// Mitsubishi GX Developer project: 12-201_1204051130   PLC: FX1N

PROGRAM MAIN
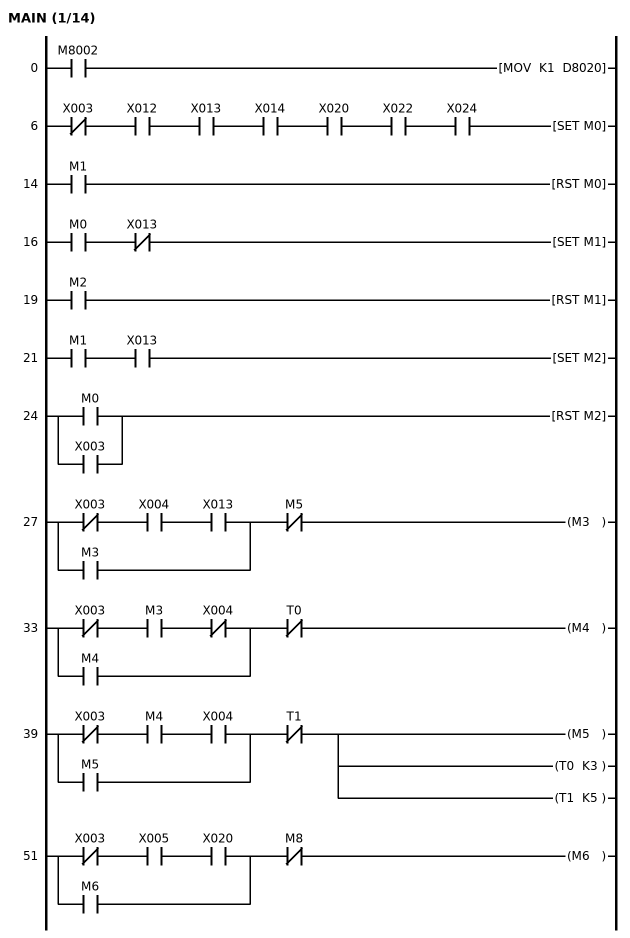
0     LD      M8002
      MOV     K1 D8020
6     LDI     X003
      AND     X012
      AND     X013
      AND     X014
      AND     X020
      AND     X022
      AND     X024
      SET     M0
14    LD      M1
      RST     M0
16    LD      M0
      ANI     X013
      SET     M1
19    LD      M2
      RST     M1
21    LD      M1
      AND     X013
      SET     M2
24    LD      M0
      OR      X003
      RST     M2
27    LDI     X003
      AND     X004
      AND     X013
      OR      M3
      ANI     M5
      OUT     M3
33    LDI     X003
      AND     M3
      ANI     X004
      OR      M4
      ANI     T0
      OUT     M4
39    LDI     X003
      AND     M4
      AND     X004
      OR      M5
      ANI     T1
      OUT     M5
      OUT     T0 K3
      OUT     T1 K5
51    LDI     X003
      AND     X005
      AND     X020
      OR      M6
      ANI     M8
      OUT     M6
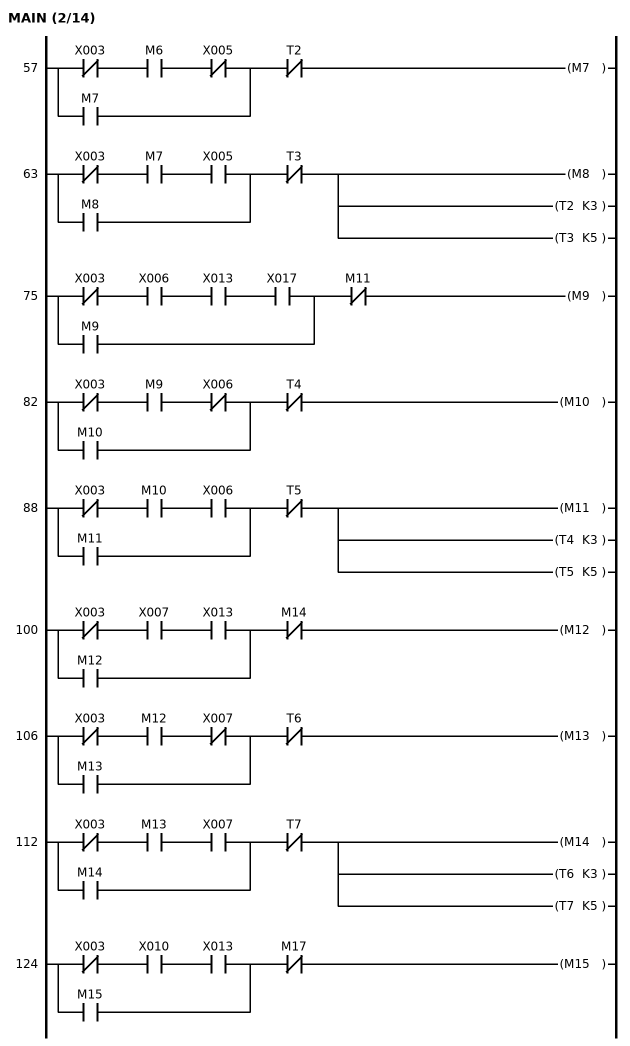
57    LDI     X003
      AND     M6
      ANI     X005
      OR      M7
      ANI     T2
      OUT     M7
63    LDI     X003
      AND     M7
      AND     X005
      OR      M8
      ANI     T3
      OUT     M8
      OUT     T2 K3
      OUT     T3 K5
75    LDI     X003
      AND     X006
      AND     X013
      AND     X017
      OR      M9
      ANI     M11
      OUT     M9
82    LDI     X003
      AND     M9
      ANI     X006
      OR      M10
      ANI     T4
      OUT     M10
88    LDI     X003
      AND     M10
      AND     X006
      OR      M11
      ANI     T5
      OUT     M11
      OUT     T4 K3
      OUT     T5 K5
100   LDI     X003
      AND     X007
      AND     X013
      OR      M12
      ANI     M14
      OUT     M12
106   LDI     X003
      AND     M12
      ANI     X007
      OR      M13
      ANI     T6
      OUT     M13
112   LDI     X003
      AND     M13
      AND     X007
      OR      M14
      ANI     T7
      OUT     M14
      OUT     T6 K3
      OUT     T7 K5
124   LDI     X003
      AND     X010
      AND     X013
      OR      M15
      ANI     M17
      OUT     M15
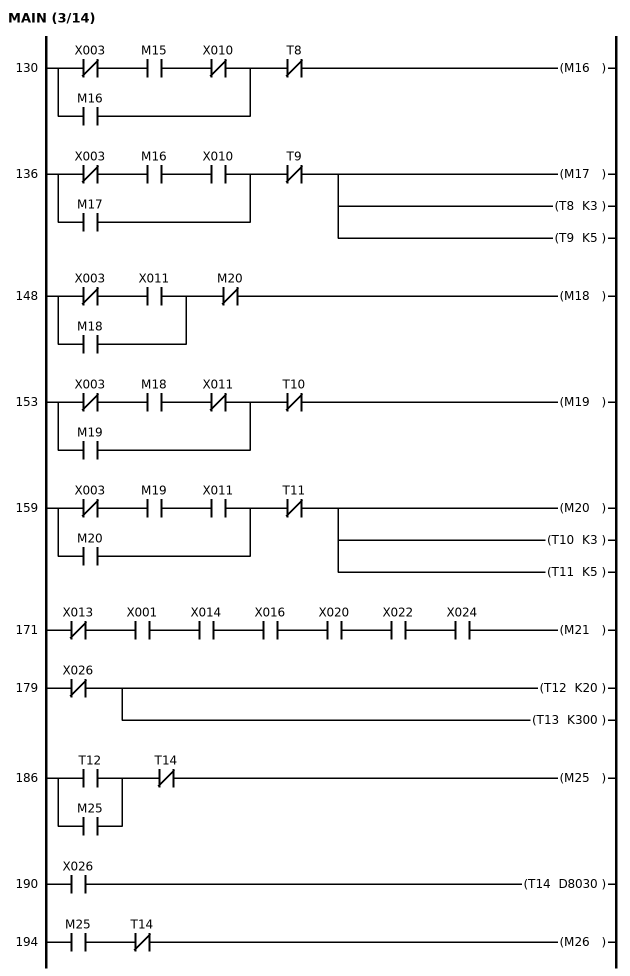
130   LDI     X003
      AND     M15
      ANI     X010
      OR      M16
      ANI     T8
      OUT     M16
136   LDI     X003
      AND     M16
      AND     X010
      OR      M17
      ANI     T9
      OUT     M17
      OUT     T8 K3
      OUT     T9 K5
148   LDI     X003
      AND     X011
      OR      M18
      ANI     M20
      OUT     M18
153   LDI     X003
      AND     M18
      ANI     X011
      OR      M19
      ANI     T10
      OUT     M19
159   LDI     X003
      AND     M19
      AND     X011
      OR      M20
      ANI     T11
      OUT     M20
      OUT     T10 K3
      OUT     T11 K5
171   LDI     X013
      AND     X001
      AND     X014
      AND     X016
      AND     X020
      AND     X022
      AND     X024
      OUT     M21
179   LDI     X026
      OUT     T12 K20
      OUT     T13 K300
186   LD      T12
      OR      M25
      ANI     T14
      OUT     M25
190   LD      X026
      OUT     T14 D8030
194   LD      M25
      ANI     T14
      OUT     M26
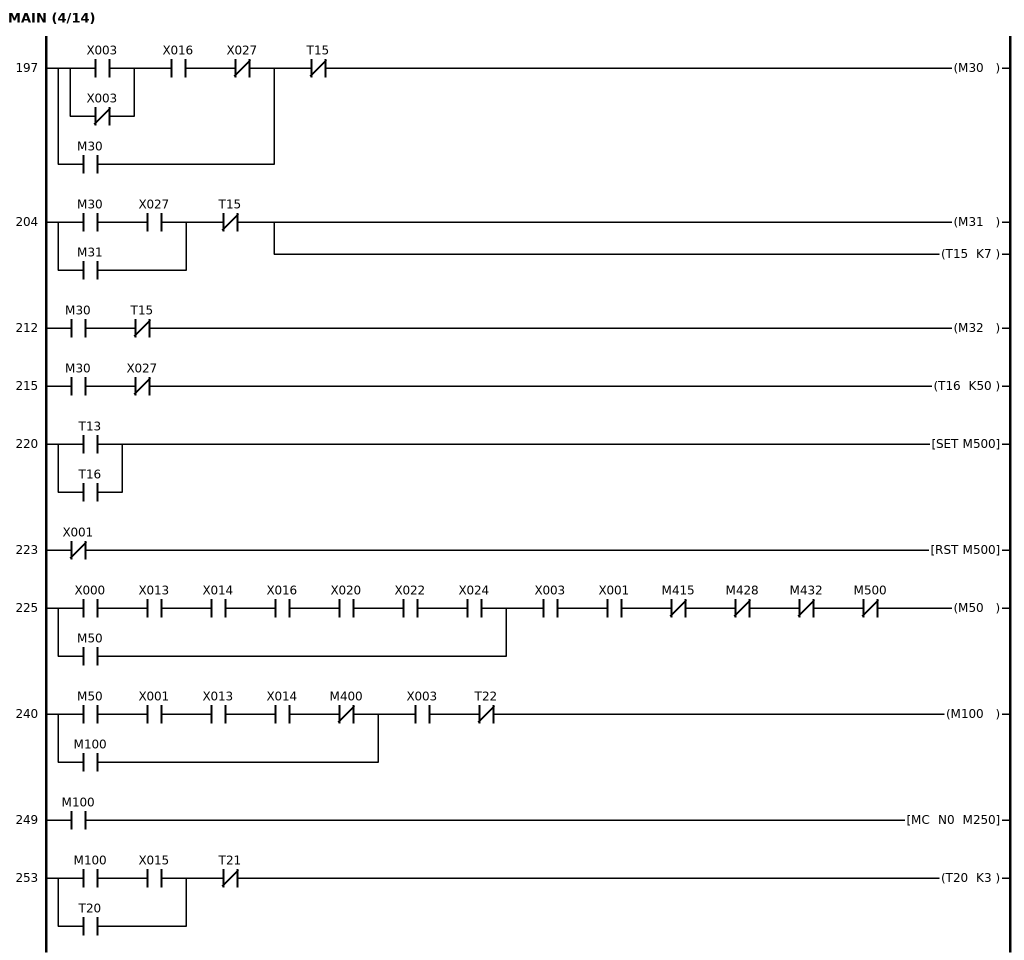
197   LD      X003
      ORI     X003
      AND     X016
      ANI     X027
      OR      M30
      ANI     T15
      OUT     M30
204   LD      M30
      AND     X027
      OR      M31
      ANI     T15
      OUT     M31
      OUT     T15 K7
212   LD      M30
      ANI     T15
      OUT     M32
215   LD      M30
      ANI     X027
      OUT     T16 K50
220   LD      T13
      OR      T16
      SET     M500
223   LDI     X001
      RST     M500
225   LD      X000
      AND     X013
      AND     X014
      AND     X016
      AND     X020
      AND     X022
      AND     X024
      OR      M50
      AND     X003
      AND     X001
      ANI     M415
      ANI     M428
      ANI     M432
      ANI     M500
      OUT     M50
240   LD      M50
      AND     X001
      AND     X013
      AND     X014
      ANI     M400
      OR      M100
      AND     X003
      ANI     T22
      OUT     M100
249   LD      M100
      MC      N0 M250
253   LD      M100
      AND     X015
      OR      T20
      ANI     T21
      OUT     T20 K3
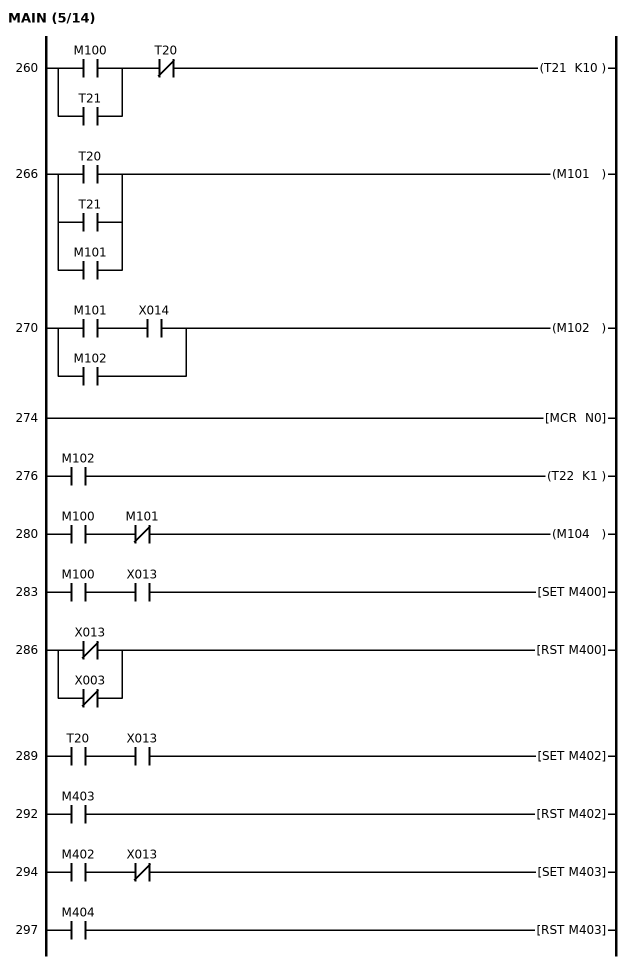
260   LD      M100
      OR      T21
      ANI     T20
      OUT     T21 K10
266   LD      T20
      OR      T21
      OR      M101
      OUT     M101
270   LD      M101
      AND     X014
      OR      M102
      OUT     M102
274   MCR     N0
276   LD      M102
      OUT     T22 K1
280   LD      M100
      ANI     M101
      OUT     M104
283   LD      M100
      AND     X013
      SET     M400
286   LDI     X013
      ORI     X003
      RST     M400
289   LD      T20
      AND     X013
      SET     M402
292   LD      M403
      RST     M402
294   LD      M402
      ANI     X013
      SET     M403
297   LD      M404
      RST     M403
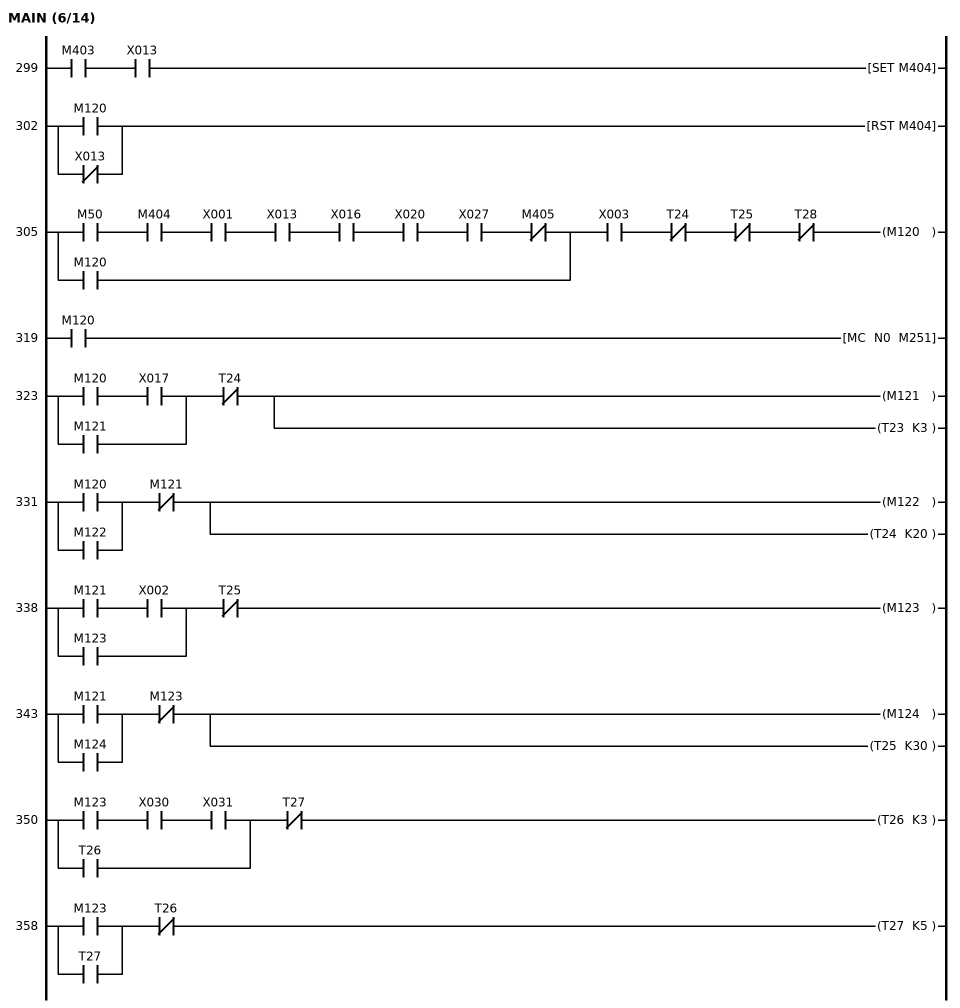
299   LD      M403
      AND     X013
      SET     M404
302   LD      M120
      ORI     X013
      RST     M404
305   LD      M50
      AND     M404
      AND     X001
      AND     X013
      AND     X016
      AND     X020
      AND     X027
      ANI     M405
      OR      M120
      AND     X003
      ANI     T24
      ANI     T25
      ANI     T28
      OUT     M120
319   LD      M120
      MC      N0 M251
323   LD      M120
      AND     X017
      OR      M121
      ANI     T24
      OUT     M121
      OUT     T23 K3
331   LD      M120
      OR      M122
      ANI     M121
      OUT     M122
      OUT     T24 K20
338   LD      M121
      AND     X002
      OR      M123
      ANI     T25
      OUT     M123
343   LD      M121
      OR      M124
      ANI     M123
      OUT     M124
      OUT     T25 K30
350   LD      M123
      AND     X030
      AND     X031
      OR      T26
      ANI     T27
      OUT     T26 K3
358   LD      M123
      OR      T27
      ANI     T26
      OUT     T27 K5
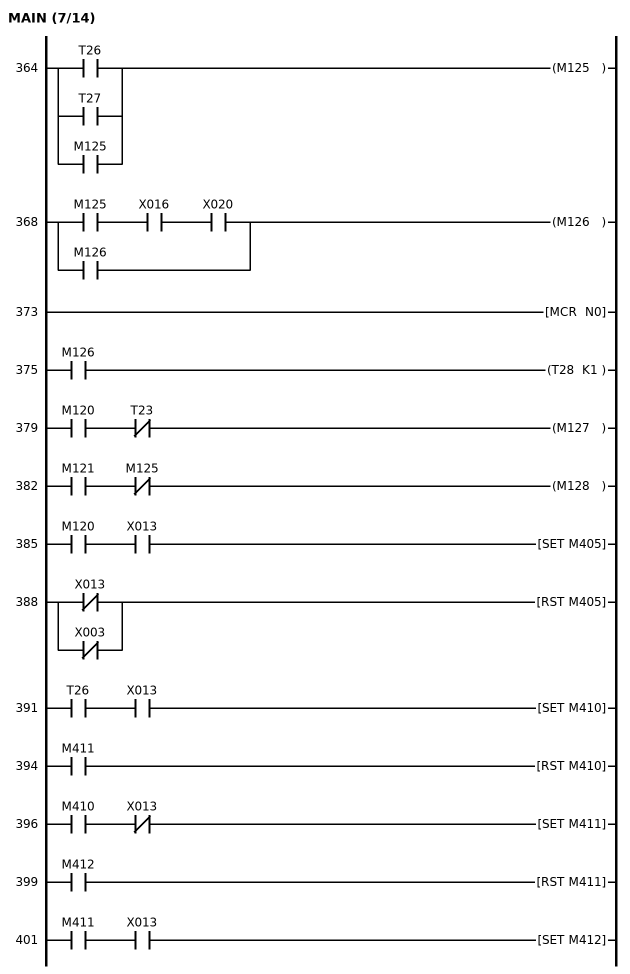
364   LD      T26
      OR      T27
      OR      M125
      OUT     M125
368   LD      M125
      AND     X016
      AND     X020
      OR      M126
      OUT     M126
373   MCR     N0
375   LD      M126
      OUT     T28 K1
379   LD      M120
      ANI     T23
      OUT     M127
382   LD      M121
      ANI     M125
      OUT     M128
385   LD      M120
      AND     X013
      SET     M405
388   LDI     X013
      ORI     X003
      RST     M405
391   LD      T26
      AND     X013
      SET     M410
394   LD      M411
      RST     M410
396   LD      M410
      ANI     X013
      SET     M411
399   LD      M412
      RST     M411
401   LD      M411
      AND     X013
      SET     M412
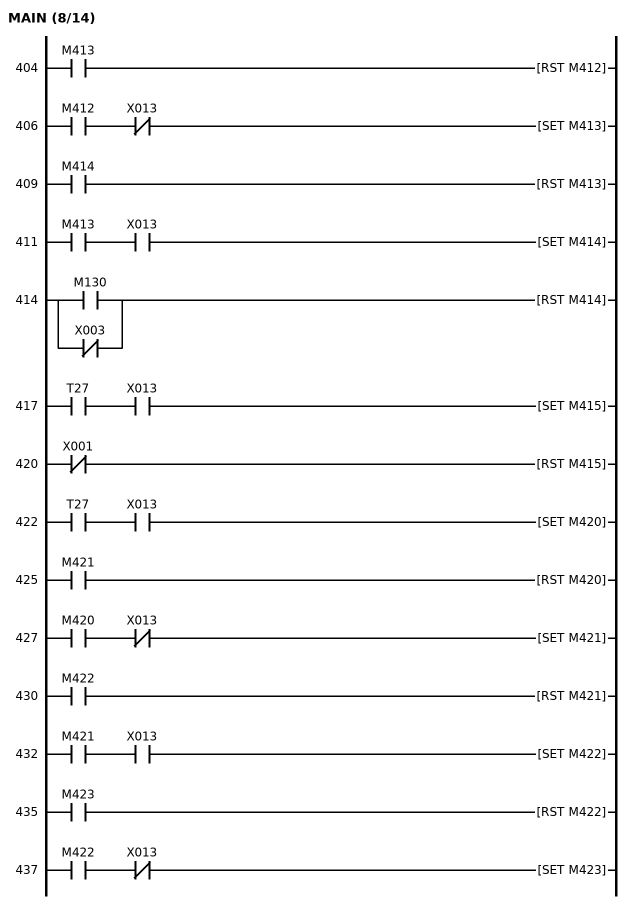
404   LD      M413
      RST     M412
406   LD      M412
      ANI     X013
      SET     M413
409   LD      M414
      RST     M413
411   LD      M413
      AND     X013
      SET     M414
414   LD      M130
      ORI     X003
      RST     M414
417   LD      T27
      AND     X013
      SET     M415
420   LDI     X001
      RST     M415
422   LD      T27
      AND     X013
      SET     M420
425   LD      M421
      RST     M420
427   LD      M420
      ANI     X013
      SET     M421
430   LD      M422
      RST     M421
432   LD      M421
      AND     X013
      SET     M422
435   LD      M423
      RST     M422
437   LD      M422
      ANI     X013
      SET     M423
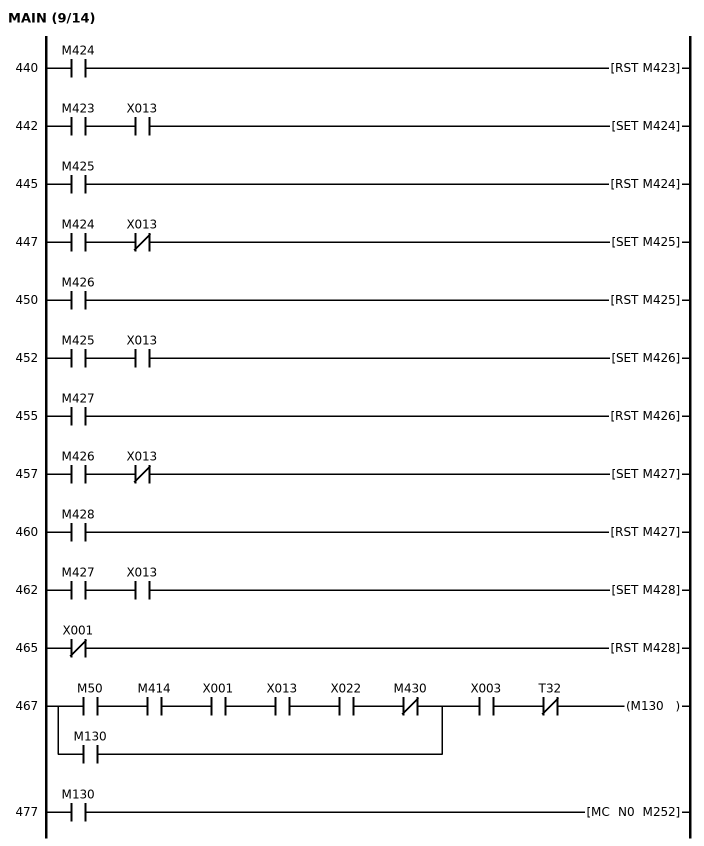
440   LD      M424
      RST     M423
442   LD      M423
      AND     X013
      SET     M424
445   LD      M425
      RST     M424
447   LD      M424
      ANI     X013
      SET     M425
450   LD      M426
      RST     M425
452   LD      M425
      AND     X013
      SET     M426
455   LD      M427
      RST     M426
457   LD      M426
      ANI     X013
      SET     M427
460   LD      M428
      RST     M427
462   LD      M427
      AND     X013
      SET     M428
465   LDI     X001
      RST     M428
467   LD      M50
      AND     M414
      AND     X001
      AND     X013
      AND     X022
      ANI     M430
      OR      M130
      AND     X003
      ANI     T32
      OUT     M130
477   LD      M130
      MC      N0 M252
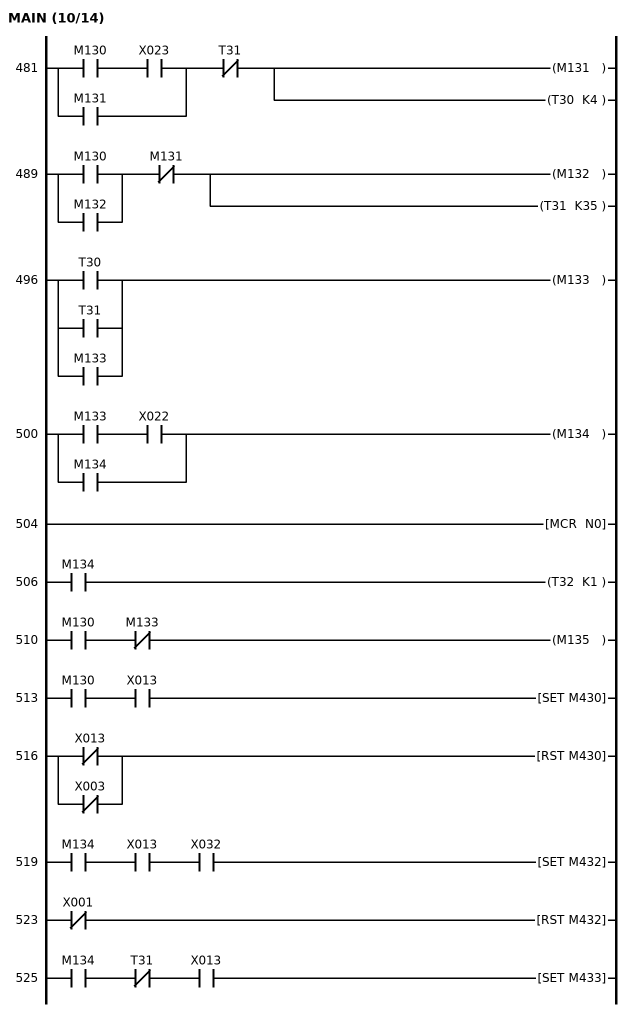
481   LD      M130
      AND     X023
      OR      M131
      ANI     T31
      OUT     M131
      OUT     T30 K4
489   LD      M130
      OR      M132
      ANI     M131
      OUT     M132
      OUT     T31 K35
496   LD      T30
      OR      T31
      OR      M133
      OUT     M133
500   LD      M133
      AND     X022
      OR      M134
      OUT     M134
504   MCR     N0
506   LD      M134
      OUT     T32 K1
510   LD      M130
      ANI     M133
      OUT     M135
513   LD      M130
      AND     X013
      SET     M430
516   LDI     X013
      ORI     X003
      RST     M430
519   LD      M134
      AND     X013
      AND     X032
      SET     M432
523   LDI     X001
      RST     M432
525   LD      M134
      ANI     T31
      AND     X013
      SET     M433
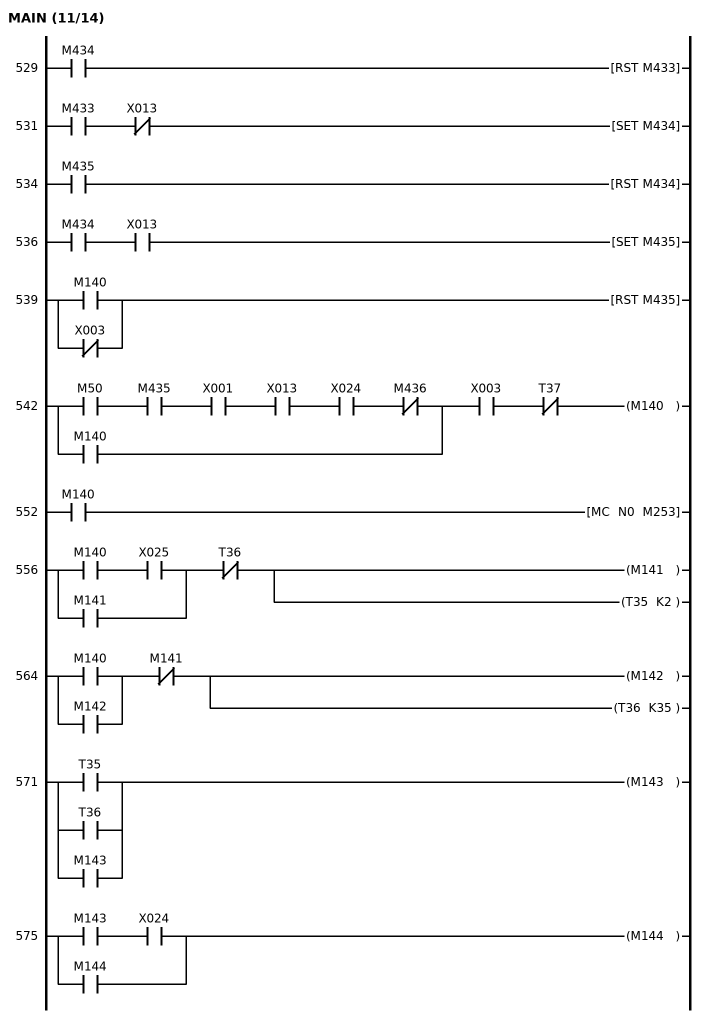
529   LD      M434
      RST     M433
531   LD      M433
      ANI     X013
      SET     M434
534   LD      M435
      RST     M434
536   LD      M434
      AND     X013
      SET     M435
539   LD      M140
      ORI     X003
      RST     M435
542   LD      M50
      AND     M435
      AND     X001
      AND     X013
      AND     X024
      ANI     M436
      OR      M140
      AND     X003
      ANI     T37
      OUT     M140
552   LD      M140
      MC      N0 M253
556   LD      M140
      AND     X025
      OR      M141
      ANI     T36
      OUT     M141
      OUT     T35 K2
564   LD      M140
      OR      M142
      ANI     M141
      OUT     M142
      OUT     T36 K35
571   LD      T35
      OR      T36
      OR      M143
      OUT     M143
575   LD      M143
      AND     X024
      OR      M144
      OUT     M144
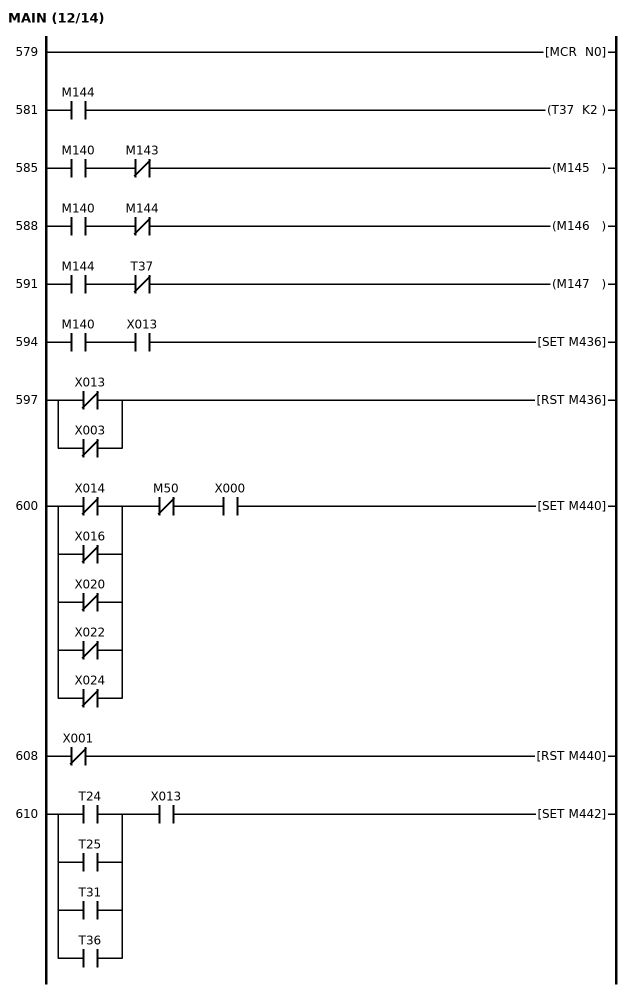
579   MCR     N0
581   LD      M144
      OUT     T37 K2
585   LD      M140
      ANI     M143
      OUT     M145
588   LD      M140
      ANI     M144
      OUT     M146
591   LD      M144
      ANI     T37
      OUT     M147
594   LD      M140
      AND     X013
      SET     M436
597   LDI     X013
      ORI     X003
      RST     M436
600   LDI     X014
      ORI     X016
      ORI     X020
      ORI     X022
      ORI     X024
      ANI     M50
      AND     X000
      SET     M440
608   LDI     X001
      RST     M440
610   LD      T24
      OR      T25
      OR      T31
      OR      T36
      AND     X013
      SET     M442
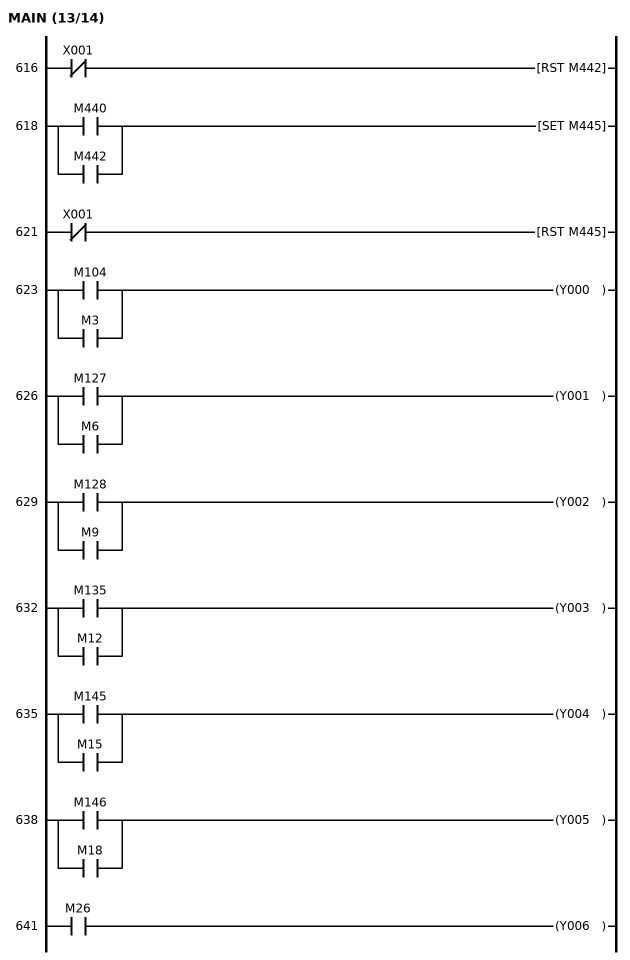
616   LDI     X001
      RST     M442
618   LD      M440
      OR      M442
      SET     M445
621   LDI     X001
      RST     M445
623   LD      M104
      OR      M3
      OUT     Y000
626   LD      M127
      OR      M6
      OUT     Y001
629   LD      M128
      OR      M9
      OUT     Y002
632   LD      M135
      OR      M12
      OUT     Y003
635   LD      M145
      OR      M15
      OUT     Y004
638   LD      M146
      OR      M18
      OUT     Y005
641   LD      M26
      OUT     Y006
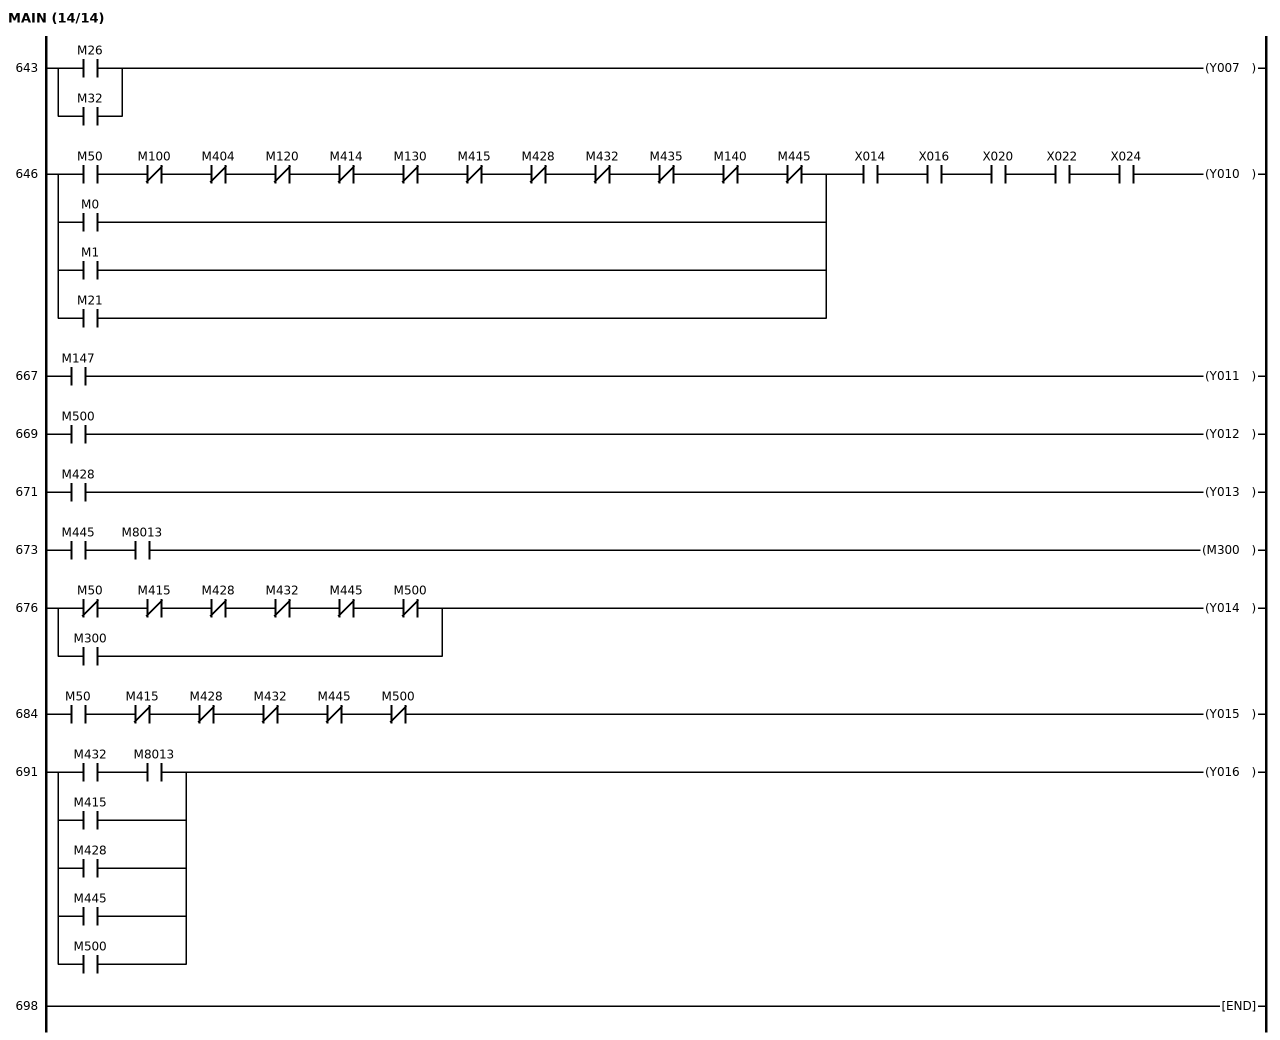
643   LD      M26
      OR      M32
      OUT     Y007
646   LD      M50
      ANI     M100
      ANI     M404
      ANI     M120
      ANI     M414
      ANI     M130
      ANI     M415
      ANI     M428
      ANI     M432
      ANI     M435
      ANI     M140
      ANI     M445
      OR      M0
      OR      M1
      OR      M21
      AND     X014
      AND     X016
      AND     X020
      AND     X022
      AND     X024
      OUT     Y010
667   LD      M147
      OUT     Y011
669   LD      M500
      OUT     Y012
671   LD      M428
      OUT     Y013
673   LD      M445
      AND     M8013
      OUT     M300
676   LDI     M50
      ANI     M415
      ANI     M428
      ANI     M432
      ANI     M445
      ANI     M500
      OR      M300
      OUT     Y014
684   LD      M50
      ANI     M415
      ANI     M428
      ANI     M432
      ANI     M445
      ANI     M500
      OUT     Y015
691   LD      M432
      AND     M8013
      OR      M415
      OR      M428
      OR      M445
      OR      M500
      OUT     Y016
698   END
END_PROGRAM
